{attribute 'TcGenerated'}
{attribute 'no-analysis'}
{attribute 'linkalways'}
// This function has been automatically generated from the project information.
VAR_GLOBAL CONSTANT
	{attribute 'const_non_replaced'}
	stLibVersion_TcTcpUdpRT : ST_LibVersion := (iMajor := 1, iMinor := 3, iBuild := 1, iRevision := 0, nFlags := 0, sVersion := '1.3.1.0');
END_VAR

(* stored: Version 1.1.0.1
   GVL Global_Version: Id {d416bef4-bd8a-0e5b-39da-1ef92f1d2fe6} *)
